PROGRAM MAIN
VAR
	fbRobot		: FB_Robot;
END_VAR

fbRobot.Cycle();

END_PROGRAM

(* stored: Version 1.1.0.1
   POU MAIN: Id {11809be1-9ff7-4a89-9e92-b65f67881044}, SpecialFunc None *)
